TYPE (* DataPanel Modules with low IO density DO Struct + Source Address *)
  (* Version 1.0, 2026-05-28, franz *)
  PACKAGE DataPanel::io::LO::DQ;
  IMPORT DataPanel::io::LO::DQ::DataPanel_LO_DO::InvalidL;
  IMPORT DataPanel::io::LO::const::LO::LO_00;
  IMPORT eclipse4diac::core::TypeHash;
  DataPanel_LO_DO_S_Single_SA : STRUCT
    u8SAMember : USINT := LO_00; (* Node SA 217..224 *)
    Port : DataPanel::io::LO::DQ::DataPanel_LO_DO_S := InvalidL; (* Identify the Port 1A..4B *)
  END_STRUCT;
END_TYPE
